FUNCTION_BLOCK E_TONOF (* standard timer function block (on/off-delay timing) *)
  (* Standard: 61499-2; Classification: standard timer function block; Description: Copyright (c) 2024 HR Agrartechnik GmbH This program and the accompanying materials are made available under the terms of the Eclipse Public License 2.0 which is available at https://www.eclipse.org/legal/epl-2.0/ SPDX-License-Identifier: EPL-2.0 *)
  (* Version 1.0, 2024-03-04, Franz Hoepfinger, HR Agrartechnik GmbH *)
  (* Version 1.1, 2024-04-23, Franz Hoepfinger, HR Agrartechnik GmbH, Add a Reset to Timer FBs *)
  (* Version 3.0, 2025-04-14, Patrick Aigner, changed package *)
  PACKAGE iec61499::events::timers;
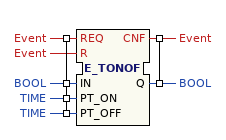
  EVENT_INPUT
    REQ WITH IN, PT_ON, PT_OFF; (* Normal Execution Request *)
    R; (* Reset *)
  END_EVENT
  EVENT_OUTPUT
    CNF WITH Q; (* Execution Confirmation *)
  END_EVENT
  VAR_INPUT
    IN : BOOL; (* Input *)
    PT_ON : TIME; (* Process time ON Delay *)
    PT_OFF : TIME; (* Process time OFF Delay *)
  END_VAR
  VAR_OUTPUT
    Q : BOOL; (* Output *)
  END_VAR
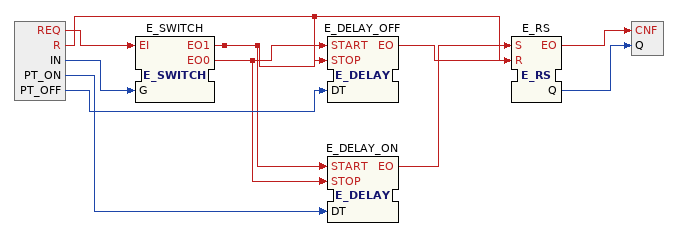
  FBS
    E_SWITCH : iec61499::events::E_SWITCH;
    E_DELAY_ON : iec61499::events::E_DELAY;
    E_RS : iec61499::events::E_RS;
    E_DELAY_OFF : iec61499::events::E_DELAY;
  END_FBS
  EVENT_CONNECTIONS
    REQ TO E_SWITCH.EI;
    E_SWITCH.EO1 TO E_DELAY_ON.START;
    E_SWITCH.EO0 TO E_DELAY_ON.STOP;
    E_DELAY_ON.EO TO E_RS.S;
    E_RS.EO TO CNF;
    E_DELAY_OFF.EO TO E_RS.R;
    E_SWITCH.EO0 TO E_DELAY_OFF.START;
    E_SWITCH.EO1 TO E_DELAY_OFF.STOP;
    R TO E_RS.R;
    R TO E_DELAY_OFF.STOP;
  END_CONNECTIONS
  DATA_CONNECTIONS
    IN TO E_SWITCH.G;
    PT_ON TO E_DELAY_ON.DT;
    E_RS.Q TO Q;
    PT_OFF TO E_DELAY_OFF.DT;
  END_CONNECTIONS
END_FUNCTION_BLOCK
